// TIA Portal V19 export
FUNCTION_BLOCK "Temperature_Control"   // FB3, LAD
{ S7_Optimized_Access := 'TRUE' }
// stored: MemoryReserve 100, SetENOAutomatically false
   VAR_INPUT
      Enable : Bool;
      Man_Enable { ExternalAccessible := 'False'; ExternalVisible := 'False'; ExternalWritable := 'False'} : Bool;
      "Temperature Sensor" : Real;
      "Process Values" : Array[0..1] of Real;
      "Simmer offset" : Real;
      "steam mode" : Int;
      "Setpoint Temperature" : Real;
      "hold time" : Time;
      "Enable temperature Hold" : Bool;
      "manual SP" : Real;
      Jacket : Bool;
   END_VAR
   VAR_OUTPUT
      "Main Valve" : Bool;
      "Simmer Valve" : Bool;
      "Stage Completed" : Bool;
      Running : Bool;
      "Enable Valve" : Bool;
      "Holding Temperature" : Bool;
      "runtime Remaining" : Real;
      "HMI Set Runtime" : Time;
      "HMI Remaining Runtime" : Time;
   END_VAR
   VAR
      "Main Valve SP" : Real;
      "Main Valve SP Reached" : Bool;
      IEC_Timer_0_Instance { S7_SetPoint := 'True'} : TON_TIME;
      IEC_Timer_0_Instance_1 { S7_SetPoint := 'True'} : TON_TIME;
      "Hold Time Completed" : Bool;
      "Reming Time" : DInt;
      Conv_Runtime : Real;
      Runtime : DInt;
      Conv_Runtime2 : Real;
      Remaingtime_1 : Real;
      Remaingtime_2 : Real;
      IEC_Timer_0_Instance_2 { S7_SetPoint := 'True'} : TON_TIME;
      "Main Valve SP Reset" { S7_SetPoint := 'True'} : Real;
      "simmer temperature" : Real;
   END_VAR
   VAR_TEMP   // added for the SCL form of the ladder/FBD networks
      _w1 : Bool;
      _w2 : Bool;
   END_VAR
BEGIN

REGION Network 1
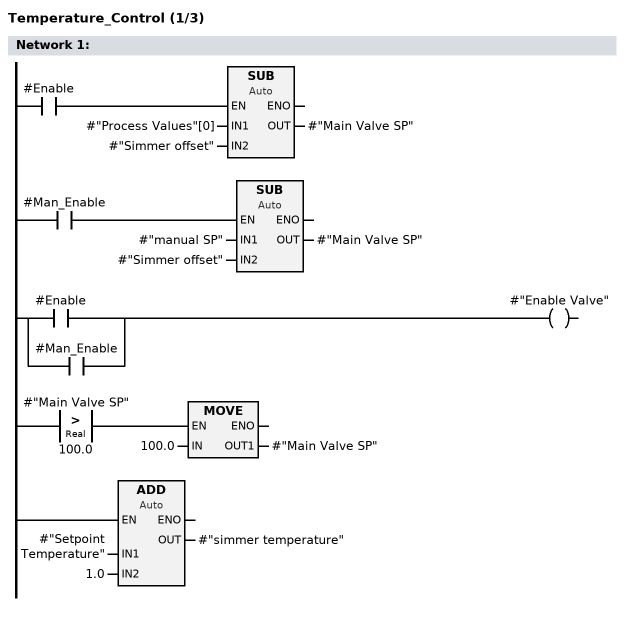
   RUNG wire#powerrail
      Contact( #Enable )
      Sub(in1 := #"Process Values"[0], in2 := #"Simmer offset", out => #"Main Valve SP")
   END_RUNG
   RUNG wire#powerrail
      Contact( #Man_Enable )
      Sub(in1 := #"manual SP", in2 := #"Simmer offset", out => #"Main Valve SP")
   END_RUNG
   RUNG wire#powerrail
      Contact( #Enable )
      wire#w1
      Coil( #"Enable Valve" )
   END_RUNG
   RUNG wire#powerrail
      Contact( #Man_Enable )
   END_RUNG wire#w1
   RUNG wire#powerrail
      { S7_Templates := "SrcType := Real" } GT_Contact(in1 := #"Main Valve SP", in2 := 100.0)
      Move(in := 100.0, out1 => #"Main Valve SP")
   END_RUNG
   RUNG wire#powerrail
      Add(in1 := #"Setpoint Temperature", in2 := 1.0, out => #"simmer temperature")
   END_RUNG
   // the same network as SCL:
   IF #Enable THEN #"Main Valve SP" := #"Process Values"[0] - #"Simmer offset"; END_IF;
   IF #Man_Enable THEN #"Main Valve SP" := #"manual SP" - #"Simmer offset"; END_IF;
   #"Enable Valve" := #Enable OR #Man_Enable;
   IF #"Main Valve SP" > 100.0 THEN #"Main Valve SP" := 100.0; END_IF;
   #"simmer temperature" := #"Setpoint Temperature" + 1.0;
END_REGION

REGION Network 2
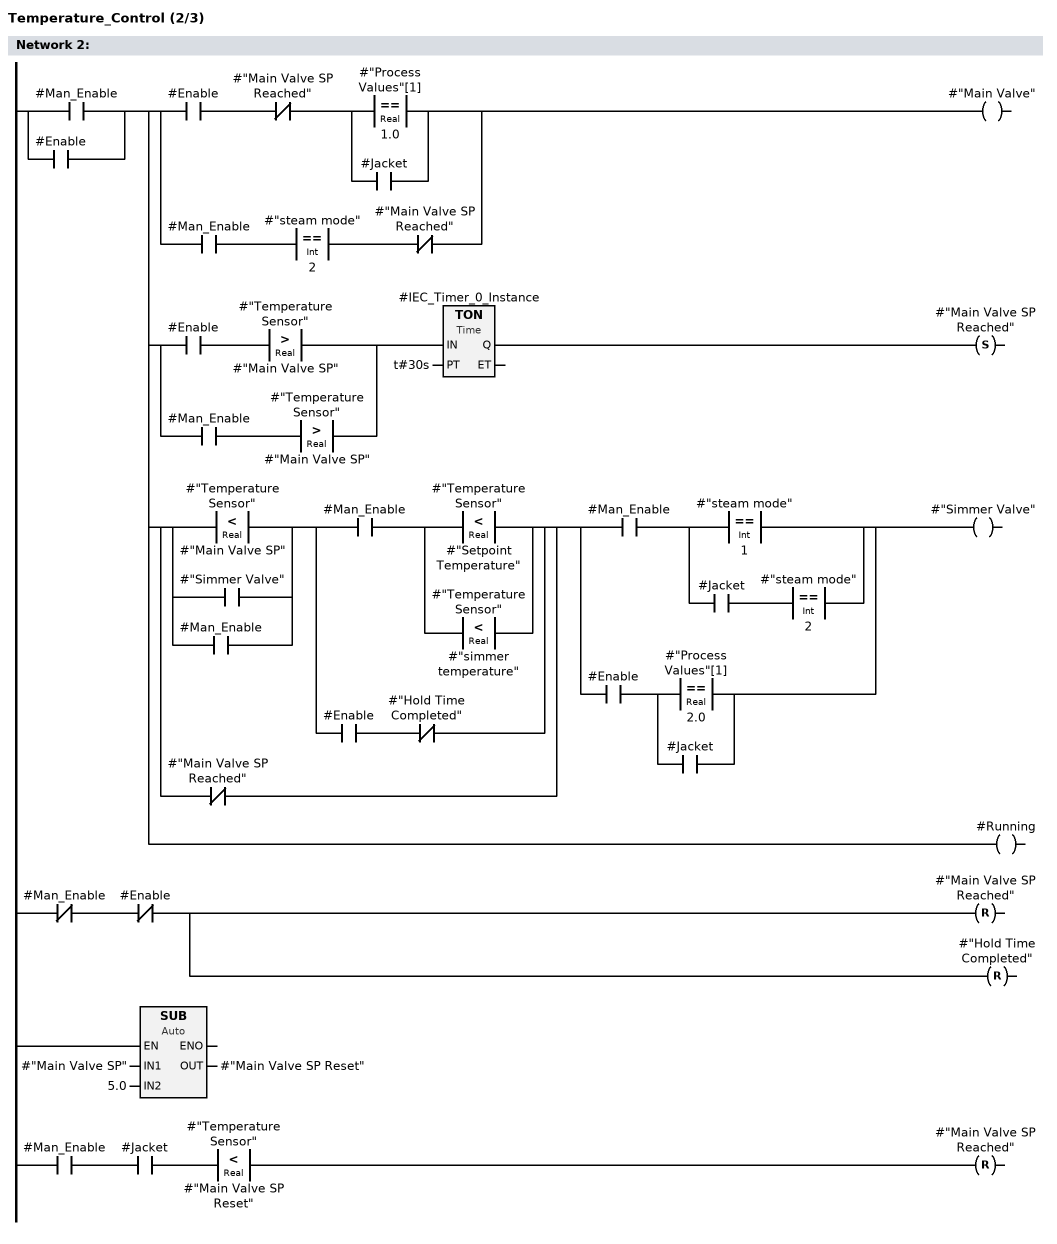
   RUNG wire#powerrail
      Contact( #Man_Enable )
      wire#w1
      Contact( #Enable )
      I_Contact( #"Main Valve SP Reached" )
      wire#w2
      { S7_Templates := "SrcType := Real" } EQ_Contact(in1 := #"Process Values"[1], in2 := 1.0)
      wire#w3
      Coil( #"Main Valve" )
   END_RUNG
   RUNG wire#powerrail
      Contact( #Enable )
   END_RUNG wire#w1
   RUNG wire#w2
      Contact( #Jacket )
   END_RUNG wire#w3
   RUNG wire#w1
      Contact( #Man_Enable )
      { S7_Templates := "SrcType := Int" } EQ_Contact(in1 := #"steam mode", in2 := 2)
      I_Contact( #"Main Valve SP Reached" )
   END_RUNG wire#w3
   RUNG wire#w1
      Contact( #Enable )
      { S7_Templates := "SrcType := Real" } GT_Contact(in1 := #"Temperature Sensor", in2 := #"Main Valve SP")
      wire#w4
      { S7_Templates := "time_type := Time" } #IEC_Timer_0_Instance.TON(pt := t#30s, et =>)
      S_Coil( #"Main Valve SP Reached" )
   END_RUNG
   RUNG wire#w1
      Contact( #Man_Enable )
      { S7_Templates := "SrcType := Real" } GT_Contact(in1 := #"Temperature Sensor", in2 := #"Main Valve SP")
   END_RUNG wire#w4
   RUNG wire#w1
      { S7_Templates := "SrcType := Real" } LT_Contact(in1 := #"Temperature Sensor", in2 := #"Main Valve SP")
      wire#w5
      Contact( #Man_Enable )
      wire#w6
      { S7_Templates := "SrcType := Real" } LT_Contact(in1 := #"Temperature Sensor", in2 := #"Setpoint Temperature")
      wire#w7
      Contact( #Man_Enable )
      wire#w8
      { S7_Templates := "SrcType := Int" } EQ_Contact(in1 := #"steam mode", in2 := 1)
      wire#w9
      Coil( #"Simmer Valve" )
   END_RUNG
   RUNG wire#w1
      Contact( #"Simmer Valve" )
   END_RUNG wire#w5
   RUNG wire#w1
      Contact( #Man_Enable )
   END_RUNG wire#w5
   RUNG wire#w6
      { S7_Templates := "SrcType := Real" } LT_Contact(in1 := #"Temperature Sensor", in2 := #"simmer temperature")
   END_RUNG wire#w7
   RUNG wire#w5
      Contact( #Enable )
      I_Contact( #"Hold Time Completed" )
   END_RUNG wire#w7
   RUNG wire#w1
      I_Contact( #"Main Valve SP Reached" )
   END_RUNG wire#w7
   RUNG wire#w8
      Contact( #Jacket )
      { S7_Templates := "SrcType := Int" } EQ_Contact(in1 := #"steam mode", in2 := 2)
   END_RUNG wire#w9
   RUNG wire#w7
      Contact( #Enable )
      wire#w10
      { S7_Templates := "SrcType := Real" } EQ_Contact(in1 := #"Process Values"[1], in2 := 2.0)
   END_RUNG wire#w9
   RUNG wire#w10
      Contact( #Jacket )
   END_RUNG wire#w9
   RUNG wire#w1
      Coil( #Running )
   END_RUNG
   RUNG wire#powerrail
      I_Contact( #Man_Enable )
      I_Contact( #Enable )
      wire#w11
      R_Coil( #"Main Valve SP Reached" )
   END_RUNG
   RUNG wire#w11
      R_Coil( #"Hold Time Completed" )
   END_RUNG
   RUNG wire#powerrail
      Sub(in1 := #"Main Valve SP", in2 := 5.0, out => #"Main Valve SP Reset")
   END_RUNG
   RUNG wire#powerrail
      Contact( #Man_Enable )
      Contact( #Jacket )
      { S7_Templates := "SrcType := Real" } LT_Contact(in1 := #"Temperature Sensor", in2 := #"Main Valve SP Reset")
      R_Coil( #"Main Valve SP Reached" )
   END_RUNG
   // the same network as SCL:
   #_w1 := #Man_Enable OR #Enable;
   #"Main Valve" := #_w1 AND ((#Enable AND NOT #"Main Valve SP Reached" AND ((#"Process Values"[1] = 1.0) OR #Jacket)) OR (#Man_Enable AND (#"steam mode" = 2) AND NOT #"Main Valve SP Reached"));
   #IEC_Timer_0_Instance(IN := #_w1 AND ((#Enable AND (#"Temperature Sensor" > #"Main Valve SP")) OR (#Man_Enable AND (#"Temperature Sensor" > #"Main Valve SP"))),   // TON
                         PT := t#30s);
   IF #IEC_Timer_0_Instance.Q THEN #"Main Valve SP Reached" := TRUE; END_IF;
   #"Simmer Valve" := #_w1 AND ((((#"Temperature Sensor" < #"Main Valve SP") OR #"Simmer Valve" OR #Man_Enable) AND ((#Man_Enable AND ((#"Temperature Sensor" < #"Setpoint Temperature") OR (#"Temperature Sensor" < #"simmer temperature"))) OR (#Enable AND NOT #"Hold Time Completed"))) OR NOT #"Main Valve SP Reached") AND ((#Man_Enable AND ((#"steam mode" = 1) OR (#Jacket AND (#"steam mode" = 2)))) OR (#Enable AND ((#"Process Values"[1] = 2.0) OR #Jacket)));
   #Running := #_w1;
   IF NOT #Man_Enable AND NOT #Enable THEN
       #"Main Valve SP Reached" := FALSE;
       #"Hold Time Completed" := FALSE;
   END_IF;
   #"Main Valve SP Reset" := #"Main Valve SP" - 5.0;
   IF #Man_Enable AND #Jacket AND (#"Temperature Sensor" < #"Main Valve SP Reset") THEN
       #"Main Valve SP Reached" := FALSE;
   END_IF;
END_REGION

REGION Network 3
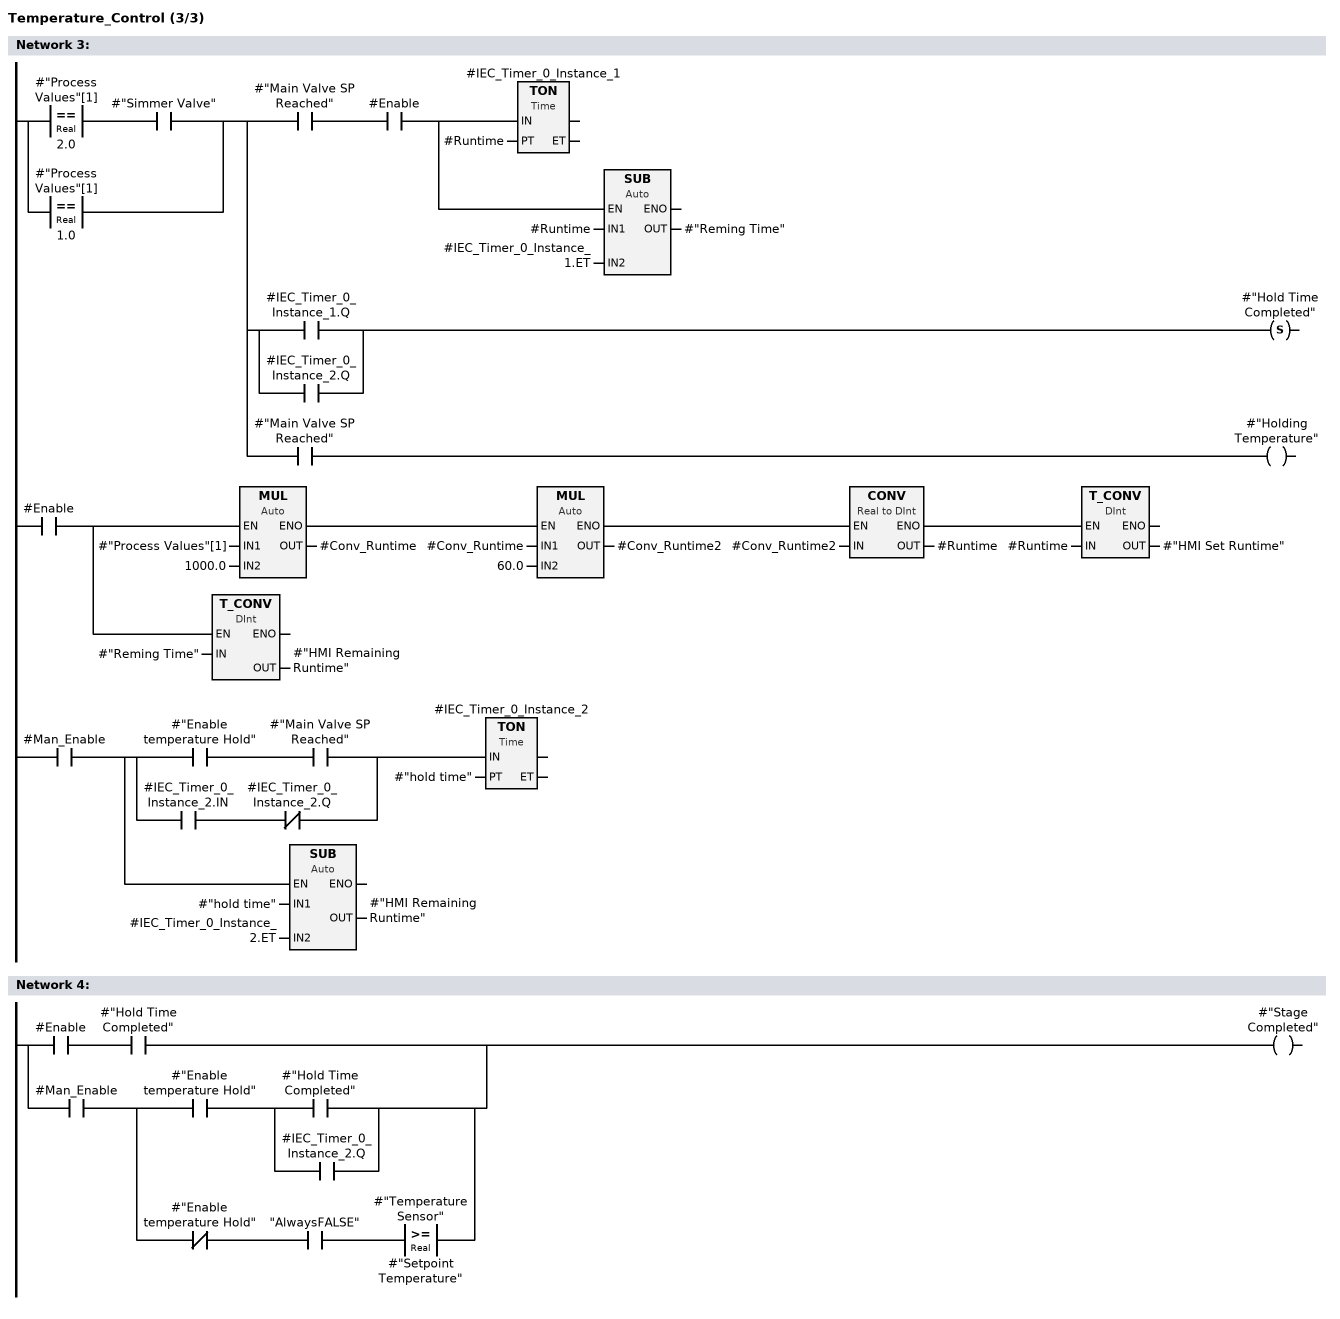
   RUNG wire#powerrail
      { S7_Templates := "SrcType := Real" } EQ_Contact(in1 := #"Process Values"[1], in2 := 2.0)
      Contact( #"Simmer Valve" )
      wire#w1
      Contact( #"Main Valve SP Reached" )
      Contact( #Enable )
      wire#w2
      { S7_Templates := "time_type := Time" } #IEC_Timer_0_Instance_1.TON(pt := #Runtime, et =>)
   END_RUNG
   RUNG wire#powerrail
      { S7_Templates := "SrcType := Real" } EQ_Contact(in1 := #"Process Values"[1], in2 := 1.0)
   END_RUNG wire#w1
   RUNG wire#w2
      Sub(in1 := #Runtime, in2 := #IEC_Timer_0_Instance_1.ET, out => #"Reming Time")
   END_RUNG
   RUNG wire#w1
      Contact( #IEC_Timer_0_Instance_1.Q )
      wire#w3
      S_Coil( #"Hold Time Completed" )
   END_RUNG
   RUNG wire#w1
      Contact( #IEC_Timer_0_Instance_2.Q )
   END_RUNG wire#w3
   RUNG wire#w1
      Contact( #"Main Valve SP Reached" )
      Coil( #"Holding Temperature" )
   END_RUNG
   RUNG wire#powerrail
      Contact( #Enable )
      wire#w4
      Mul(in1 := #"Process Values"[1], in2 := 1000.0, out => #Conv_Runtime)
      Mul(in1 := #Conv_Runtime, in2 := 60.0, out => #Conv_Runtime2)
      { S7_Templates := "[SrcType := Real, DestType := DInt]" } Convert(in := #Conv_Runtime2, out => #Runtime)
      { S7_Templates := "[src_type := DInt, dest_type := Time]" } T_CONV(IN := #Runtime, OUT => #"HMI Set Runtime")
   END_RUNG
   RUNG wire#w4
      { S7_Templates := "[src_type := DInt, dest_type := Time]" } T_CONV(IN := #"Reming Time", OUT => #"HMI Remaining Runtime")
   END_RUNG
   RUNG wire#powerrail
      Contact( #Man_Enable )
      wire#w5
      Contact( #"Enable temperature Hold" )
      Contact( #"Main Valve SP Reached" )
      wire#w6
      { S7_Templates := "time_type := Time" } #IEC_Timer_0_Instance_2.TON(pt := #"hold time", et =>)
   END_RUNG
   RUNG wire#w5
      Contact( #IEC_Timer_0_Instance_2.IN )
      I_Contact( #IEC_Timer_0_Instance_2.Q )
   END_RUNG wire#w6
   RUNG wire#w5
      Sub(in1 := #"hold time", in2 := #IEC_Timer_0_Instance_2.ET, out => #"HMI Remaining Runtime")
   END_RUNG
   // the same network as SCL:
   #_w1 := ((#"Process Values"[1] = 2.0) AND #"Simmer Valve") OR (#"Process Values"[1] = 1.0);
   #_w2 := #_w1 AND #"Main Valve SP Reached" AND #Enable;
   #IEC_Timer_0_Instance_1(IN := #_w2, PT := #Runtime);   // TON
   IF #_w2 THEN #"Reming Time" := #Runtime - #IEC_Timer_0_Instance_1.ET; END_IF;
   IF #_w1 AND (#IEC_Timer_0_Instance_1.Q OR #IEC_Timer_0_Instance_2.Q) THEN
       #"Hold Time Completed" := TRUE;
   END_IF;
   #"Holding Temperature" := #_w1 AND #"Main Valve SP Reached";
   IF #Enable THEN
       #Conv_Runtime := #"Process Values"[1] * 1000.0;
       #Conv_Runtime2 := #Conv_Runtime * 60.0;
       #Runtime := REAL_TO_DINT(#Conv_Runtime2);
       T_CONV(IN := #Runtime, OUT => #"HMI Set Runtime");
       T_CONV(IN := #"Reming Time", OUT => #"HMI Remaining Runtime");
   END_IF;
   #IEC_Timer_0_Instance_2(IN := #Man_Enable AND ((#"Enable temperature Hold" AND #"Main Valve SP Reached") OR (#IEC_Timer_0_Instance_2.IN AND NOT #IEC_Timer_0_Instance_2.Q)),   // TON
                           PT := #"hold time");
   IF #Man_Enable THEN #"HMI Remaining Runtime" := #"hold time" - #IEC_Timer_0_Instance_2.ET; END_IF;
END_REGION

REGION Network 4
   RUNG wire#powerrail
      Contact( #Enable )
      Contact( #"Hold Time Completed" )
      wire#w1
      Coil( #"Stage Completed" )
   END_RUNG
   RUNG wire#powerrail
      Contact( #Man_Enable )
      wire#w2
      Contact( #"Enable temperature Hold" )
      wire#w3
      Contact( #"Hold Time Completed" )
   END_RUNG wire#w1
   RUNG wire#w3
      Contact( #IEC_Timer_0_Instance_2.Q )
   END_RUNG wire#w1
   RUNG wire#w2
      I_Contact( #"Enable temperature Hold" )
      Contact( "AlwaysFALSE" )
      { S7_Templates := "SrcType := Real" } GE_Contact(in1 := #"Temperature Sensor", in2 := #"Setpoint Temperature")
   END_RUNG wire#w1
   // the same network as SCL:
   #"Stage Completed" := (#Enable AND #"Hold Time Completed") OR (#Man_Enable AND ((#"Enable temperature Hold" AND (#"Hold Time Completed" OR #IEC_Timer_0_Instance_2.Q)) OR (NOT #"Enable temperature Hold" AND "AlwaysFALSE" AND (#"Temperature Sensor" >= #"Setpoint Temperature"))));
END_REGION
END_FUNCTION_BLOCK
